{attribute addProperty BoxType "EK1100-0000-0018"}
{attribute addProperty Id "Beckhoff_EL68xxEK1122Beckhoff_EL68xxEK1122_833CFEA0162A_0001_EL6851_0000_0017EL6851_527AC90F4298537.25A_0002_EL6851_0000_0018EL6851_527AC90F4298537.25A_0003_EL6851_0000_0019EL6851_527AC90F4298537.25A_0004_EL6851_0000_0020EL6851_077DD54E4298537.25A_0005_EL6851_0000_0021EL6851_077DD54E4298537.25A_0006_EL6851_0010_0016EL6851_41B974CF65882.25A_0007_EL6851_0010_0017EL6851_41B974CF65882.25A_0008_EL6851_0010_0018EL6851_41B974CF65882.25A_0009_EL6851_0010_0019EL6851_20762A1865882.25A_0010_EL6861_0000_0016EL6861_B662EC3C2162270.25A_0011_EL6861_0000_0017EL6861_B662EC3C2162270.25"}
{attribute addProperty CRC "770402349"}
{attribute addProperty SizeInBites "28462"}
{attribute addProperty SizeInBytes "3557.75"}
TYPE Beckhoff_EL68xx_2DEB682D EXTENDS EK1100_179A0949 :
STRUCT
	{attribute addProperty Name "Beckhoff_EL68xxEK1122"}
	Beckhoff_EL68xxEK1122 : Beckhoff_EL68xxEK1122_833CFEA0;
	{attribute addProperty Name "A_0001_EL6851_0000_0017"}
	A_0001_EL6851_0000_0017 : EL6851_527AC90F;
	{attribute addProperty Name "A_0002_EL6851_0000_0018"}
	A_0002_EL6851_0000_0018 : EL6851_527AC90F;
	{attribute addProperty Name "A_0003_EL6851_0000_0019"}
	A_0003_EL6851_0000_0019 : EL6851_527AC90F;
	{attribute addProperty Name "A_0004_EL6851_0000_0020"}
	A_0004_EL6851_0000_0020 : EL6851_077DD54E;
	{attribute addProperty Name "A_0005_EL6851_0000_0021"}
	A_0005_EL6851_0000_0021 : EL6851_077DD54E;
	{attribute addProperty Name "A_0006_EL6851_0010_0016"}
	A_0006_EL6851_0010_0016 : EL6851_41B974CF;
	{attribute addProperty Name "A_0007_EL6851_0010_0017"}
	A_0007_EL6851_0010_0017 : EL6851_41B974CF;
	{attribute addProperty Name "A_0008_EL6851_0010_0018"}
	A_0008_EL6851_0010_0018 : EL6851_41B974CF;
	{attribute addProperty Name "A_0009_EL6851_0010_0019"}
	A_0009_EL6851_0010_0019 : EL6851_20762A18;
	{attribute addProperty Name "A_0010_EL6861_0000_0016"}
	A_0010_EL6861_0000_0016 : EL6861_B662EC3C;
	{attribute addProperty Name "A_0011_EL6861_0000_0017"}
	A_0011_EL6861_0000_0017 : EL6861_B662EC3C;
END_STRUCT
END_TYPE

(* stored: Version 1.2.0.0, ProductVersion 3.1.4024.9
   DUT Beckhoff_EL68xx_2DEB682D: Id {edb1b221-13bb-445e-9d1d-d68d82e5e163} *)
